RoboDK station: Stringer C-Top1-BOX1.rdk

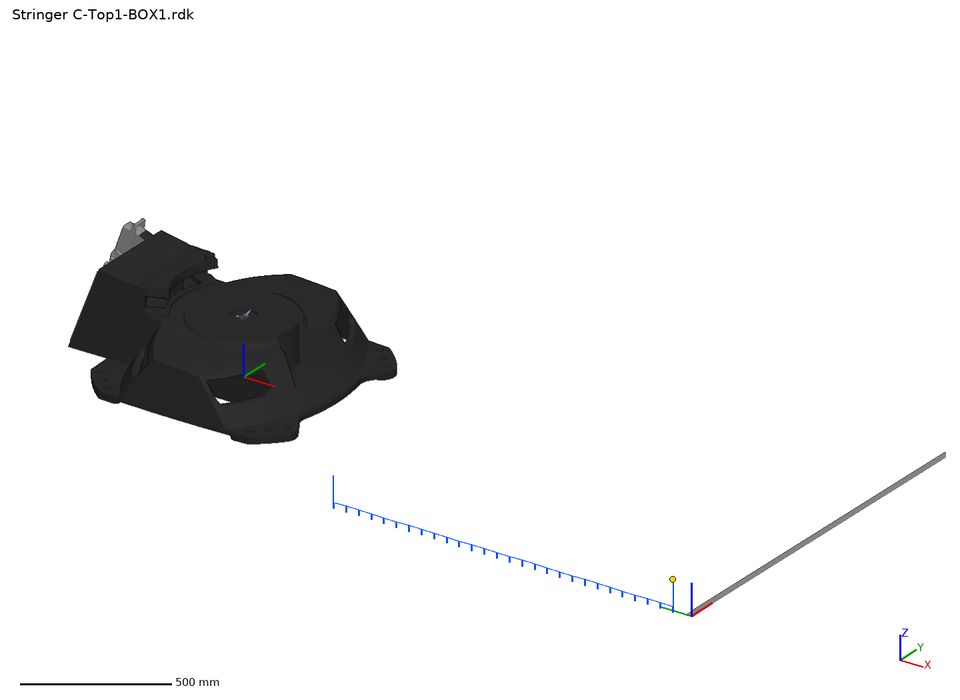
[picture v0: the station drawn from its stored meshes, robots at their saved joint values, targets as dots, program paths as lines]
Station Stringer C-Top1-BOX1 (saved by RoboDK 5.2.3). Poses are relative to the parent item; angles as X-Y-Z fixed-axis rotations.
  - frame KUKA KR 210 R2700 extra Base at (0, 0, 0) mm
    - robot KUKA KR 210 R2700 extra: 6 axes, payload 210 kg, reach 2696 mm, repeatability 0.06 mm, weight 1068 kg
        joint limits [-185, -140, -120, -350, -125, -350] to [185, -5, 155, 350, 125, 350]; home [0, -90, 90, 0, 0, 0]; saved at [-43.372, -23.234, 76.99, 78.17, 26.203, -113.146]
      - tool Spindle, TCP at (32, 0, 260) mm, rotated rx 0 ry 39 rz 0 deg, size 157.3 x 72 x 259.9 mm
  - frame Frame 2 at (1800, 0, -372.68) mm, rotated rx 0 ry 0 rz 90 deg
    - object L-Stringer C - Top1-BOX1 at (0, 0, 0) mm, size 1455.7 x 20 x 20 mm, geometry from L-Stringer C - Top1-BOX1.stl
    - object Stringer C-Top1-BOX1 at (0, 0, 0) mm, rotated rx 0 ry 0 rz -90 deg, 28 curves, geometry from Point 28
  - machining project Point settings: rotZ(0) | rotX(0)*rotY(0) | rotz(0) | onStart | onPathStart | onApproach | onPoint | onRetract | onFinish | SetRPM(%1) | SetTool(%1) | Extruder(%1) | default | default | OutOnMov(%1) | OutOffMov(%1) | onPathFinish | M_RunCode(%1)
  - program Point (151 instructions, listed below)
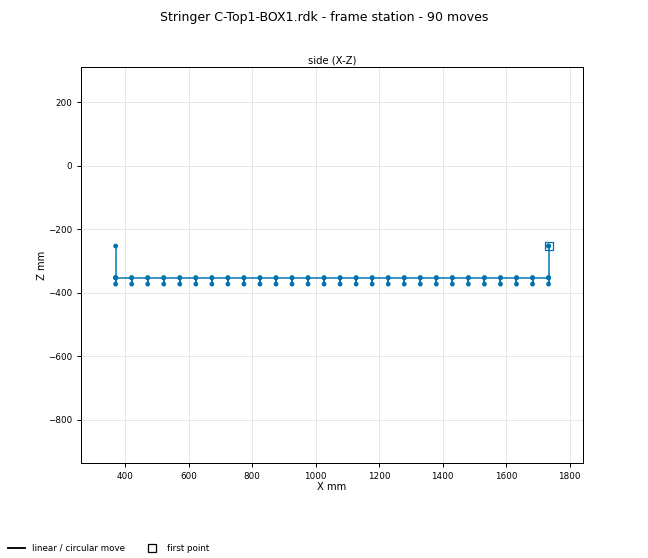
[picture p0: tool path of Stringer C-Top1-BOX1.rdk in frame station, 90 of 90 moves have a stored position in this frame; points joined in program order, loops and branches not executed]

--- program Point (robot KUKA KR 210 R2700 extra) ---
  Smooth(1)
  Set speed (1000.0 mm/s)
  Set Ref.: Frame 2
  Set Tool: Spindle
  Show Spindle
  MoveJ 1 to (-11.7, 66.57, 120) mm, rotated rx -180 ry 0 rz -180 deg; joints [-2.517, -34.017, 111.866, 176.493, 26.866, -178.828]
  MoveL 2 to (-11.7, 66.57, 120) mm, rotated rx -180 ry 0 rz -180 deg; joints [-2.517, -34.017, 111.866, 176.493, 26.866, -178.828]
  MoveL 3 to (-11.7, 66.57, 20) mm, rotated rx -180 ry 0 rz -180 deg; joints [-2.517, -28.686, 109.223, 176.787, 29.549, -179.161]
  MoveL 4 to (-11.7, 66.57, 20) mm, rotated rx -180 ry 0 rz -180 deg; joints [-2.517, -28.686, 109.223, 176.787, 29.549, -179.161]
  Set speed (50.0 mm/s)
  MoveL 5 to (-11.7, 66.57, 0) mm, rotated rx -180 ry 0 rz -180 deg; joints [-2.517, -27.628, 108.647, 176.834, 30.03, -179.215]
  MoveL 6 to (-11.7, 66.57, 20) mm, rotated rx -180 ry 0 rz -180 deg; joints [-2.517, -28.686, 109.223, 176.787, 29.549, -179.161]
  Set speed (1000.0 mm/s)
  MoveL 7 to (-11.7, 117.09, 20) mm, rotated rx -180 ry 0 rz -180 deg; joints [-4.422, -28.665, 109.064, 174.334, 29.436, -178.501]
  Set speed (50.0 mm/s)
  MoveL 8 to (-11.7, 117.09, 0) mm, rotated rx -180 ry 0 rz -180 deg; joints [-4.422, -27.608, 108.489, 174.417, 29.915, -178.596]
  MoveL 9 to (-11.7, 117.09, 20) mm, rotated rx -180 ry 0 rz -180 deg; joints [-4.422, -28.665, 109.064, 174.334, 29.436, -178.501]
  Set speed (1000.0 mm/s)
  MoveL 10 to (-11.7, 167.61, 20) mm, rotated rx -180 ry 0 rz -180 deg; joints [-6.316, -28.631, 108.818, 171.858, 29.264, -177.802]
  Set speed (50.0 mm/s)
  MoveL 11 to (-11.7, 167.61, 0) mm, rotated rx -180 ry 0 rz -180 deg; joints [-6.316, -27.576, 108.244, 171.977, 29.739, -177.939]
  MoveL 12 to (-11.7, 167.61, 20) mm, rotated rx -180 ry 0 rz -180 deg; joints [-6.316, -28.631, 108.818, 171.858, 29.264, -177.802]
  Set speed (1000.0 mm/s)
  MoveL 13 to (-11.7, 218.13, 20) mm, rotated rx 180 ry 0 rz 180 deg; joints [-8.197, -28.583, 108.485, 169.346, 29.035, -177.048]
  Set speed (50.0 mm/s)
  MoveL 14 to (-11.7, 218.13, 0) mm, rotated rx -180 ry 0 rz -180 deg; joints [-8.197, -27.532, 107.912, 169.503, 29.506, -177.227]
  MoveL 15 to (-11.7, 218.13, 20) mm, rotated rx 180 ry 0 rz 180 deg; joints [-8.197, -28.583, 108.485, 169.346, 29.035, -177.048]
  Set speed (1000.0 mm/s)
  MoveL 16 to (-11.7, 268.65, 20) mm, rotated rx 180 ry 0 rz -180 deg; joints [-10.06, -28.522, 108.066, 166.789, 28.754, -176.221]
  Set speed (50.0 mm/s)
  MoveL 17 to (-11.7, 268.65, 0) mm, rotated rx 180 ry 0 rz 180 deg; joints [-10.06, -27.474, 107.494, 166.984, 29.217, -176.444]
  MoveL 18 to (-11.7, 268.65, 20) mm, rotated rx 180 ry 0 rz -180 deg; joints [-10.06, -28.522, 108.066, 166.789, 28.754, -176.221]
  Set speed (1000.0 mm/s)
  MoveL 19 to (-11.7, 319.16, 20) mm, rotated rx 180 ry 0 rz 180 deg; joints [-11.902, -28.445, 107.56, 164.177, 28.424, -175.307]
  Set speed (50.0 mm/s)
  MoveL 20 to (-11.7, 319.16, 0) mm, rotated rx 180 ry 0 rz -180 deg; joints [-11.902, -27.401, 106.99, 164.411, 28.88, -175.574]
  MoveL 21 to (-11.7, 319.16, 20) mm, rotated rx 180 ry 0 rz 180 deg; joints [-11.902, -28.445, 107.56, 164.177, 28.424, -175.307]
  Set speed (1000.0 mm/s)
  MoveL 22 to (-11.7, 369.68, 20) mm, rotated rx 180 ry 0 rz 180 deg; joints [-13.72, -28.35, 106.967, 161.495, 28.052, -174.288]
  Set speed (50.0 mm/s)
  MoveL 23 to (-11.7, 369.68, 0) mm, rotated rx 180 ry 0 rz 180 deg; joints [-13.72, -27.312, 106.399, 161.771, 28.498, -174.6]
  MoveL 24 to (-11.7, 369.68, 20) mm, rotated rx 180 ry 0 rz 180 deg; joints [-13.72, -28.35, 106.967, 161.495, 28.052, -174.288]
  Set speed (1000.0 mm/s)
  MoveL 25 to (-11.7, 420.2, 20) mm, rotated rx 180 ry 0 rz -180 deg; joints [-15.509, -28.237, 106.289, 158.735, 27.644, -173.148]
  Set speed (50.0 mm/s)
  MoveL 26 to (-11.7, 420.2, 0) mm, rotated rx -180 ry 0 rz -180 deg; joints [-15.509, -27.205, 105.724, 159.053, 28.079, -173.507]
  MoveL 27 to (-11.7, 420.2, 20) mm, rotated rx 180 ry 0 rz -180 deg; joints [-15.509, -28.237, 106.289, 158.735, 27.644, -173.148]
  Set speed (1000.0 mm/s)
  MoveL 28 to (-11.7, 470.72, 20) mm, rotated rx 180 ry 0 rz 180 deg; joints [-17.268, -28.104, 105.526, 155.883, 27.207, -171.872]
  Set speed (50.0 mm/s)
  MoveL 29 to (-11.7, 470.72, 0) mm, rotated rx -180 ry 0 rz -180 deg; joints [-17.268, -27.078, 104.962, 156.245, 27.629, -172.279]
  MoveL 30 to (-11.7, 470.72, 20) mm, rotated rx 180 ry 0 rz 180 deg; joints [-17.268, -28.104, 105.526, 155.883, 27.207, -171.872]
  Set speed (1000.0 mm/s)
  MoveL 31 to (-11.7, 521.24, 20) mm, rotated rx -180 ry 0 rz -180 deg; joints [-18.995, -27.948, 104.677, 152.928, 26.749, -170.444]
  Set speed (50.0 mm/s)
  MoveL 32 to (-11.7, 521.24, 0) mm, rotated rx -180 ry 0 rz -180 deg; joints [-18.995, -26.929, 104.116, 153.336, 27.157, -170.901]
  MoveL 33 to (-11.7, 521.24, 20) mm, rotated rx -180 ry 0 rz -180 deg; joints [-18.995, -27.948, 104.677, 152.928, 26.749, -170.444]
  Set speed (1000.0 mm/s)
  MoveL 34 to (-11.7, 571.76, 20) mm, rotated rx 180 ry 0 rz -180 deg; joints [-20.686, -27.768, 103.743, 149.86, 26.278, -168.852]
  Set speed (50.0 mm/s)
  MoveL 35 to (-11.7, 571.76, 0) mm, rotated rx -180 ry 0 rz -180 deg; joints [-20.686, -26.756, 103.185, 150.314, 26.671, -169.359]
  MoveL 36 to (-11.7, 571.76, 20) mm, rotated rx 180 ry 0 rz -180 deg; joints [-20.686, -27.768, 103.743, 149.86, 26.278, -168.852]
  Set speed (1000.0 mm/s)
  MoveL 37 to (-11.7, 622.28, 20) mm, rotated rx -180 ry 0 rz -180 deg; joints [-22.34, -27.561, 102.725, 146.666, 25.805, -167.081]
  Set speed (50.0 mm/s)
  MoveL 38 to (-11.7, 622.28, 0) mm, rotated rx -180 ry 0 rz -180 deg; joints [-22.34, -26.557, 102.17, 147.168, 26.181, -167.639]
  MoveL 39 to (-11.7, 622.28, 20) mm, rotated rx -180 ry 0 rz -180 deg; joints [-22.34, -27.561, 102.725, 146.666, 25.805, -167.081]
  Set speed (1000.0 mm/s)
  MoveL 40 to (-11.7, 672.79, 20) mm, rotated rx 180 ry 0 rz 180 deg; joints [-23.956, -27.326, 101.623, 143.34, 25.339, -165.121]
  Set speed (50.0 mm/s)
  MoveL 41 to (-11.7, 672.79, 0) mm, rotated rx 180 ry 0 rz -180 deg; joints [-23.956, -26.331, 101.07, 143.89, 25.695, -165.731]
  MoveL 42 to (-11.7, 672.79, 20) mm, rotated rx 180 ry 0 rz 180 deg; joints [-23.956, -27.326, 101.623, 143.34, 25.339, -165.121]
  Set speed (1000.0 mm/s)
  MoveL 43 to (-11.7, 723.31, 20) mm, rotated rx -180 ry 0 rz -180 deg; joints [-25.532, -27.061, 100.437, 139.871, 24.889, -162.963]
  Set speed (50.0 mm/s)
  MoveL 44 to (-11.7, 723.31, 0) mm, rotated rx -180 ry 0 rz -180 deg; joints [-25.532, -26.074, 99.886, 140.469, 25.225, -163.623]
  MoveL 45 to (-11.7, 723.31, 20) mm, rotated rx -180 ry 0 rz -180 deg; joints [-25.532, -27.061, 100.437, 139.871, 24.889, -162.963]
  Set speed (1000.0 mm/s)
  MoveL 46 to (-11.7, 773.83, 20) mm, rotated rx -180 ry 0 rz -180 deg; joints [-27.069, -26.763, 99.166, 136.256, 24.467, -160.6]
  Set speed (50.0 mm/s)
  MoveL 47 to (-11.7, 773.83, 0) mm, rotated rx 180 ry 0 rz 180 deg; joints [-27.069, -25.785, 98.618, 136.901, 24.78, -161.31]
  MoveL 48 to (-11.7, 773.83, 20) mm, rotated rx -180 ry 0 rz -180 deg; joints [-27.069, -26.763, 99.166, 136.256, 24.467, -160.6]
  Set speed (1000.0 mm/s)
  MoveL 49 to (-11.7, 824.35, 20) mm, rotated rx 180 ry 0 rz 180 deg; joints [-28.564, -26.431, 97.811, 132.493, 24.084, -158.031]
  Set speed (50.0 mm/s)
  MoveL 50 to (-11.7, 824.35, 0) mm, rotated rx 180 ry 0 rz -180 deg; joints [-28.564, -25.462, 97.265, 133.183, 24.372, -158.788]
  MoveL 51 to (-11.7, 824.35, 20) mm, rotated rx 180 ry 0 rz 180 deg; joints [-28.564, -26.431, 97.811, 132.493, 24.084, -158.031]
  Set speed (1000.0 mm/s)
  MoveL 52 to (-11.7, 874.87, 20) mm, rotated rx -180 ry 0 rz -180 deg; joints [-30.018, -26.062, 96.371, 128.585, 23.75, -155.258]
  Set speed (50.0 mm/s)
  MoveL 53 to (-11.7, 874.87, 0) mm, rotated rx 180 ry 0 rz -180 deg; joints [-30.018, -25.102, 95.827, 129.316, 24.012, -156.058]
  MoveL 54 to (-11.7, 874.87, 20) mm, rotated rx -180 ry 0 rz -180 deg; joints [-30.018, -26.062, 96.371, 128.585, 23.75, -155.258]
  Set speed (1000.0 mm/s)
  MoveL 55 to (-11.7, 925.39, 20) mm, rotated rx 180 ry 0 rz 180 deg; joints [-31.43, -25.655, 94.845, 124.539, 23.477, -152.289]
  Set speed (50.0 mm/s)
  MoveL 56 to (-11.7, 925.39, 0) mm, rotated rx 180 ry 0 rz -180 deg; joints [-31.43, -24.704, 94.304, 125.306, 23.711, -153.126]
  MoveL 57 to (-11.7, 925.39, 20) mm, rotated rx 180 ry 0 rz 180 deg; joints [-31.43, -25.655, 94.845, 124.539, 23.477, -152.289]
  Set speed (1000.0 mm/s)
  MoveL 58 to (-11.7, 975.91, 20) mm, rotated rx 180 ry 0 rz 180 deg; joints [-32.801, -25.207, 93.234, 120.368, 23.274, -149.137]
  Set speed (50.0 mm/s)
  MoveL 59 to (-11.7, 975.91, 0) mm, rotated rx 180 ry 0 rz -180 deg; joints [-32.801, -24.266, 92.694, 121.165, 23.479, -150.005]
  MoveL 60 to (-11.7, 975.91, 20) mm, rotated rx 180 ry 0 rz 180 deg; joints [-32.801, -25.207, 93.234, 120.368, 23.274, -149.137]
  Set speed (1000.0 mm/s)
  MoveL 61 to (-11.7, 1026.42, 20) mm, rotated rx 180 ry 0 rz 180 deg; joints [-34.131, -24.717, 91.535, 116.094, 23.153, -145.822]
  Set speed (50.0 mm/s)
  MoveL 62 to (-11.7, 1026.42, 0) mm, rotated rx 180 ry 0 rz 180 deg; joints [-34.131, -23.785, 90.996, 116.912, 23.328, -146.713]
  MoveL 63 to (-11.7, 1026.42, 20) mm, rotated rx 180 ry 0 rz 180 deg; joints [-34.131, -24.717, 91.535, 116.094, 23.153, -145.822]
  Set speed (1000.0 mm/s)
  MoveL 64 to (-11.7, 1076.94, 20) mm, rotated rx -180 ry 0 rz -180 deg; joints [-35.421, -24.182, 89.747, 111.739, 23.12, -142.37]
  Set speed (50.0 mm/s)
  MoveL 65 to (-11.7, 1076.94, 0) mm, rotated rx -180 ry 0 rz -180 deg; joints [-35.421, -23.26, 89.209, 112.569, 23.265, -143.273]
  MoveL 66 to (-11.7, 1076.94, 20) mm, rotated rx -180 ry 0 rz -180 deg; joints [-35.421, -24.182, 89.747, 111.739, 23.12, -142.37]
  Set speed (1000.0 mm/s)
  MoveL 67 to (-11.7, 1127.46, 20) mm, rotated rx -180 ry 0 rz -180 deg; joints [-36.67, -23.6, 87.868, 107.334, 23.186, -138.81]
  Set speed (50.0 mm/s)
  MoveL 68 to (-11.7, 1127.46, 0) mm, rotated rx -180 ry 0 rz -180 deg; joints [-36.67, -22.687, 87.33, 108.166, 23.3, -139.715]
  MoveL 69 to (-11.7, 1127.46, 20) mm, rotated rx -180 ry 0 rz -180 deg; joints [-36.67, -23.6, 87.868, 107.334, 23.186, -138.81]
  Set speed (1000.0 mm/s)
  MoveL 70 to (-11.7, 1177.98, 20) mm, rotated rx 180 ry 0 rz -180 deg; joints [-37.881, -22.969, 85.895, 102.911, 23.356, -135.176]
  Set speed (50.0 mm/s)
  MoveL 71 to (-11.7, 1177.98, 0) mm, rotated rx 180 ry 0 rz -180 deg; joints [-37.881, -22.065, 85.357, 103.734, 23.44, -136.072]
  MoveL 72 to (-11.7, 1177.98, 20) mm, rotated rx 180 ry 0 rz -180 deg; joints [-37.881, -22.969, 85.895, 102.911, 23.356, -135.176]
  Set speed (1000.0 mm/s)
  MoveL 73 to (-11.7, 1228.5, 20) mm, rotated rx 180 ry 0 rz 180 deg; joints [-39.052, -22.286, 83.826, 98.507, 23.635, -131.504]
  Set speed (50.0 mm/s)
  MoveL 74 to (-11.7, 1228.5, 0) mm, rotated rx -180 ry 0 rz -180 deg; joints [-39.052, -21.39, 83.286, 99.31, 23.69, -132.381]
  MoveL 75 to (-11.7, 1228.5, 20) mm, rotated rx 180 ry 0 rz 180 deg; joints [-39.052, -22.286, 83.826, 98.507, 23.635, -131.504]
  Set speed (1000.0 mm/s)
  MoveL 76 to (-11.7, 1279.02, 20) mm, rotated rx -180 ry 0 rz -180 deg; joints [-40.186, -21.549, 81.656, 94.155, 24.026, -127.829]
  Set speed (50.0 mm/s)
  MoveL 77 to (-11.7, 1279.02, 0) mm, rotated rx -180 ry 0 rz -180 deg; joints [-40.186, -20.661, 81.115, 94.928, 24.054, -128.676]
  MoveL 78 to (-11.7, 1279.02, 20) mm, rotated rx -180 ry 0 rz -180 deg; joints [-40.186, -21.549, 81.656, 94.155, 24.026, -127.829]
  Set speed (1000.0 mm/s)
  MoveL 79 to (-11.7, 1329.54, 20) mm, rotated rx 180 ry 0 rz -180 deg; joints [-41.284, -20.754, 79.381, 89.887, 24.533, -124.184]
  Set speed (50.0 mm/s)
  MoveL 80 to (-11.7, 1329.54, 0) mm, rotated rx 180 ry 0 rz 180 deg; joints [-41.284, -19.874, 78.836, 90.622, 24.535, -124.991]
  MoveL 81 to (-11.7, 1329.54, 20) mm, rotated rx 180 ry 0 rz -180 deg; joints [-41.284, -20.754, 79.381, 89.887, 24.533, -124.184]
  Set speed (1000.0 mm/s)
  MoveL 82 to (-11.7, 1380.05, 20) mm, rotated rx 180 ry 0 rz -180 deg; joints [-42.345, -19.898, 76.995, 85.733, 25.156, -120.597]
  Set speed (50.0 mm/s)
  MoveL 83 to (-11.7, 1380.05, 0) mm, rotated rx -180 ry 0 rz -180 deg; joints [-42.345, -19.025, 76.447, 86.422, 25.134, -121.358]
  MoveL 84 to (-11.7, 1380.05, 20) mm, rotated rx 180 ry 0 rz -180 deg; joints [-42.345, -19.898, 76.995, 85.733, 25.156, -120.597]
  Set speed (1000.0 mm/s)
  MoveL 85 to (-11.7, 1430.57, 20) mm, rotated rx -180 ry 0 rz 180 deg; joints [-43.372, -18.976, 74.491, 81.714, 25.896, -117.09]
  Set speed (50.0 mm/s)
  MoveL 86 to (-11.7, 1430.57, 0) mm, rotated rx -180 ry 0 rz -180 deg; joints [-43.372, -18.109, 73.937, 82.352, 25.853, -117.799]
  MoveL 87 to (-11.7, 1430.57, 20) mm, rotated rx -180 ry 0 rz 180 deg; joints [-43.372, -18.976, 74.491, 81.714, 25.896, -117.09]
  MoveL 88 to (-11.7, 1430.57, 20) mm, rotated rx -180 ry 0 rz 180 deg; joints [-43.372, -18.976, 74.491, 81.714, 25.896, -117.09]
  Set speed (1000.0 mm/s)
  MoveL 89 to (-11.7, 1430.57, 20) mm, rotated rx -180 ry 0 rz 180 deg; joints [-43.372, -18.976, 74.491, 81.714, 25.896, -117.09]
  MoveL 90 to (-11.7, 1430.57, 120) mm, rotated rx 180 ry 0 rz 180 deg; joints [-43.372, -23.234, 76.99, 78.17, 26.203, -113.146]
